Yaskawa INFORM job: TEST123.JBI

/JOB
//NAME TEST123
//POS
///NPOS 1,1,0,0,0,0
///TOOL 0
///POSTYPE ROBOT
///RECTAN
///RCONF 0,0,0,0,1,0,0,0,0,0,0,0,0,0,0,0,0,0,0,0,0,0,0,0
C00000=-108.652,-2131.032,-1243.630,-31.0513,-12.1965,-74.8063
///RCONF 0,0,0,0,0,0,0,0,0,0,0,0,0,0,0,0,0,0,0,0,0,0,0,0
BC00000=1428.669,3134.895,961.157
//INST
///DATE 2024/01/16 12:48
///ATTR SC,RW,RJ
////FRAME ROBOT
///GROUP1 RB1,BS1
NOP
MOVJ C00000 BC00000 VJ=0.78
END
